FUNCTION SquareSignal : REAL
VAR_INPUT
	r_MinValue : REAL;
	r_MaxValue : REAL;
	r_Offset : REAL;
	r_Kreisfrequenz : REAL;
	r_Time: REAL;

	
END_VAR
VAR
		r_Temp : REAL;
END_VAR

r_Temp:= SIN(r_Kreisfrequenz*r_Time); 
IF r_temp>=0 THEN
SquareSignal := r_MaxValue + r_Offset;	
ELSE
SquareSignal := r_MinValue + r_Offset;	
END_IF

END_FUNCTION

(* stored: Version 1.1.0.1, ProductVersion 3.1.4022.12
   POU SquareSignal: Id {cf83d338-9e15-44f0-9695-a17f54b52369}, SpecialFunc None *)
